(* PLC project Untitled1, Beckhoff Automation GmbH TF6420 Database Server Query Analyser 1.0.0.0 *)
(* stored: creationDateTime 2021-11-03T18:05:57, modificationDateTime 2021-11-03T18:05:57 *)

TYPE ST_Webinar : STRUCT
  ID : LINT;
  Timestamp : DT;
  AnalogValue : LREAL;
  DigitalValue : BOOL;
END_STRUCT;
END_TYPE
